Fanuc KAREL source: kf00117.KL

-- PROVISIONAL review KL for V1013-1; original PC SHA256 6c3973d947667a8ec9363725856677990920d0b3d98214dbc7c9ca9462eaf5fd
-- Incomplete behavior may be omitted. Consult companion uncertainty JSON. Do not deploy.
PROGRAM KF00117
%NOLOCKGROUP
BEGIN
  -- UNRESOLVED_PC offsets 0-1; opcodes 7B
  -- UNRESOLVED_PC offsets 6-21; opcodes 17,9D,33,34,23
  -- UNRESOLVED_PC offsets 26-30; opcodes 7F
  -- UNRESOLVED_PC offsets 35-45; opcodes 27,22,AA
  -- UNRESOLVED_PC offsets 50-54; opcodes 7F
END KF00117
